VISUALIZATION HMI_DebugCell_Stack  // 2x2
END_VISUALIZATION

(* stored: Version 1.1.0.1, ProductVersion 3.1.4022.12
   Visu HMI_DebugCell_Stack: Id {c9866237-5e64-43f2-a238-324e15549b0c} *)
